{attribute 'reflection'}
PROGRAM SystemBase // system base program, from here all modules are controlled and the system functions are called.
VAR_INPUT // System configuration settings
	bIcfAirCheckPresent	: BOOL := TRUE; // System is not equiped with air pressure sensor 
END_VAR
VAR	// Fault indications
	bMissingCond		: BOOL := FALSE ; // Module missing condition active
	bFatalFault			: BOOL := FALSE ; // Module fatal fault is active
	bCycleFault			: BOOL := FALSE ; // Module cycle fault is active

	// Check values
	bReferenceOk		: BOOL := FALSE ; // All module references  have been checked

	// State indication
	bSafeStopping		: BOOL := FALSE ; // Module is stopping by safety
	bIsSafe				: BOOL := FALSE ; // Module is safe and locked until safety is ok
	bNoreference		: BOOL := FALSE ; // Module Startup Undefined initialization required

	bInitializing		: BOOL := FALSE ; // Module startup initializing
	bInitialized		: BOOL := FALSE ; // Module startup initialized waiting for startup command
	
	bParametersLoaded 	: BOOL := FALSE ; // Parameters have been loaded from the file(s) 

	bIdle 				: BOOL := FALSE ; // Module startup Idle no commands active

	bEnabling 			: BOOL := FALSE ; // Module Startup enabeling 
	bEnabled 			: BOOL := FALSE ; // Module Startup Enabled
	
	bHoming				: BOOL := FALSE ; // Module startup homing back to base position and recalibrate
	bHomed 				: BOOL := FALSE ; // Module startup homed waiting for further further commands

	bHolding 			: BOOL := FALSE ; // Module Module Hold motion command executing
	bHeld	 			: BOOL := FALSE ; // Module Hold Motion is held until command is released	
	
	bResetting 			: BOOL := FALSE ; // Module Reset resetting error status
	bResetDone 			: BOOL := FALSE ; // Module reset is done   

	bManual 			: BOOL := FALSE ; // Module Work status Module in Manual 
	
	bStartSemiAuto		: BOOL := FALSE ; // Start semi automatic mode 
	bSemiAuto			: BOOL := FALSE ; // Module work status module in semi automatic
	
	bStartAuto			: BOOL := FALSE ; // Start automatic mode
	bAutomatic 			: BOOL := FALSE ; // Module Work status Module in Automatic mode
	bStopAuto			: BOOL := FALSE ; // Start automatic mode
	bStoppingAuto		: BOOL := FALSE ; // Start automatic mode
	
	bCmdPause			: BOOL := FALSE ; // Pause all modules 
	bPaused 			: BOOL := FALSE ; // all modules are paused
	
	bPoweringOff		: BOOL := FALSE ; // Module is powering off
	bPoweredOff			: BOOL := FALSE ; // Module has powered off 	

	bModuleLocked		: BOOL := FALSE ; // a module is locked for commands
	
	bAckWarningsBusy	: BOOL := FALSE	; // The acknowledge process is busy
END_VAR
VAR
	// System inputs 
	ibPowerSupplyOk	 	AT%I*	: BOOL  ; // System Power supply is ok 
	iSystemSafetyFault	AT%I*	: BOOL	; // System safety Fault
	fbAirpressureOk 			: Fb_DevDigitalInputFunctions  	; // system airpressure is ok
	fbCmdResetSafety		 	: FB_DevPushbuttonLight 		; // System reset
	
	fTrigPowerSupply			: F_TRIG ; // falling edge trigger for power supply
	toffMainAir					: TOF	:= (PT := T#500MS ); // Main air supply off delay
	// System safety valve
	fbValveMainAirSupply		: FB_DevValve ; // Main air supply valve 
	
	// System HMI commands
	fbStartSemiAuto				: FB_DevHMIButton ; // HMI start semi automatic button 
	fbStartAuto					: FB_DevHMIButton ; // HMI start automatic button
	fbResetSystem				: FB_DevHMIButton ; // HMI Reset system
	fbCmdPowerOff				: FB_DevHMIButton ; // HMI Power off system
	fbAckWarning				: FB_DevHMIButton ; // HMI Acknowledge warnings

	// system Commands 
	fbCmdStartSystem		 	: FB_DevPushbuttonLight  		; // (re)start system input from button
	fbCmdStartAuto				: FB_DevPushbuttonLight			; // Start system automatic cycle
	fbCmdStopAuto				: FB_DevPushbuttonLight			; // Start system automatic cycle
	
	//System state
	bSafetyOK					: BOOL := FALSE ;
	bAirOk						: BOOL := FALSE ; // Air pressure is ok 
	bSystemOK					: BOOL := FALSE ; // all safety and vitals are OK
	eStateSystem				: E_StateSystem := E_StateSystem.NoReference ; // State of system
	
	// Set system variables
	fbSetSystemVariables		: Fb_SystemVariables ;
	
	// System Fault handling
//	fbSystemFaultHandler		: Fb_SystemFaultHandler ;
//	fbOperatorMessage			: FB_OperatorMessageDisplay ; //Operator message or system state message hadler 

	// Local Fault Handling
	stFault					: UDT_Fault			; // Message data

 	// Module states
	nNumberOfModules			: UDINT := 0 ; // Number of modules added to the system 
	arpModules					: ARRAY [1..gvl_main.cnMaxNUMBEROFMODULES] OF Udt_ModuleId ; 

	// power down system function
	ntShutDown					: NT_Shutdown ; // shutdown system function 

	// Manual controller
	bDevicesAddedtoManual 		: BOOL := FALSE ; // Add system device (buttons) to manual controller
	

	// Function path 
	{attribute 'instance-path'} 
    {attribute 'noinit'}
	sPath			: STRING	; // Path name of function (used for manual reference
END_VAR
VAR // safety 
	// inputs 
	ibEstopOk 			AT%I*	: BOOL  ; // system emergency stop ok
	ibSystemSafetyOK	AT%I*	: BOOL  ; // System is safe 
	iSafetyFBErr		AT%I*	: BOOL	; // The "FB Error" group signal
	iSafetyComErr		AT%I*	: BOOL	; // The "Com Error" group signal
	iSafetyOtherErr		AT%I*	: BOOL	; // The "Other Err" group signal
	iSafetyOutErr		AT%I*	: BOOL	; // The "Out Err" group signal
	iSTOFault			AT%I* 	: BOOL	; // Motor safe torque off fault active
	
	// Outputs 
	qbSafetyErrAckn		AT%Q*	: BOOL ; // Safety error acknowledge
	qbRunSafety			AT%Q*	: BOOL ; // Run safety program
	qbResetSafety		AT%Q*	: BOOL ; // reset safety program
	qbSTOErrAckn		AT%Q*	: BOOL ; // Safet torque off error acnowledge

	// safety Reset Timer	
	TofSafetyErrAck				: TOF := (PT := T#500MS); // Safety reset timer
	TOfSTOErrAck				: TOF := (PT := T#500MS); // Safe torque off rest timer
END_VAR
VAR // Miscellaneous
	bFirstCycle : BOOL := TRUE; // Is this the first time the PRG is called?
	bPersistentDataFail	: BOOL := TRUE ;
END_VAR
VAR PERSISTENT // Persistent data check
	bPersistentFlag	: BOOL := FALSE ; // Persistent dat in tack flag
END_VAR

// Exec safety control
ExecSafetyControl();

// Call faulthandler
//fbSystemFaultHandler( 	nNumberOfModules	:= nNumberOfModules,
//						arpModules			:= arpModules,
//						bsystemInitialized	:= bInitialized,
//						bSystemFF			=> bFatalFault,
//						bSystemCF			=> bCycleFault,
//						bSystemMC			=> bMissingCond);

// Check if this is the first cycle the PRG is called
// if not, return. This is to make sure all modules are connected. 
IF bFirstCycle THEN
	bFirstCycle := FALSE;
	RETURN;
END_IF

// check system functions
IF bInitialized THEN 
	CheckSystemOK();
	CheckSystemCommands();
END_IF 

// Run system
ExecSystemRun();

// call device functions 
CallSystemFunctions();

// Call operator warning acknowledgement
ExecAckWarnings();

// Call modules 
CallModules();

METHOD PRIVATE CallModules : BOOL
VAR
	i : UDINT ;
END_VAR
VAR
	AllAutomatic : BOOL ;
	
	Stopping : BOOL;
	bAllStopped : BOOL;
END_VAR
// set base conditions
bReferenceOk	:= TRUE ;
bIsSafe			:= TRUE ;
bIdle			:= TRUE ;	
bHeld			:= TRUE ;
bResetDone 		S= bResetting	;
bManual			:= TRUE	;
bSemiAuto		:= TRUE ;
bAutomatic		:= FALSE; // Reverse feedback 
AllAutomatic 	:= TRUE ;
bStoppingAuto	:= TRUE ;
bEnabled		S= bEnabling ;
bPoweredOff		:= TRUE;
bHomed 			:= TRUE;
bPaused 		:= TRUE;
bAllStopped     := TRUE;

// copy inputs to modules 
FOR i := 1 TO nNumberOfModules DO 
	// set system commands
	arpModules[i].pFunction^.bEnable			:= bEnabled			;
	arpModules[i].pFunction^.bCmdReset			:= bResetting		;
	arpModules[i].pFunction^.bSafetyOK			:= NOT bSafeStopping;
	arpModules[i].pFunction^.bCmdPause			:= bCmdPause		; 
	// Read state indications 
	bReferenceOk 	:= arpModules[i].pFunction^.bReferenceOk 	AND bReferenceOk; 
	bIsSafe 		:= arpModules[i].pFunction^.bIsSafe 		AND bIsSafe		;
	bEnabled 		:= arpModules[i].pFunction^.bEnable 		AND bEnabled	;
	bHeld			:= arpModules[i].pFunction^.bHeld 			AND bHeld		;
	bResetDone		:= arpModules[i].pFunction^.bResetDone 		AND bResetDone	;
	bManual			:= arpModules[i].pFunction^.bManual 		AND bManual		;
	bSemiAuto		:= arpModules[i].pFunction^.bSemiAuto 		AND bSemiAuto	;
	bPoweredOff 	:= arpModules[i].pFunction^.bPoweredOff 	AND bPoweredOff	;
	bHomed			:= arpModules[i].pFunction^.bHomed			AND bHomed 		;
	bPaused			:= arpModules[i].pFunction^.bPaused			AND bPaused		;
	bModuleLocked	S= arpModules[i].pFunction^.bLocked							; // Module is locked for commnds
	bCmdPause 		R= arpModules[i].pFunction^.bReqContinue					; // Request continue from module
	bCmdPause		S= arpModules[i].pFunction^.bReqPause						; // Request for pause from module
	bAutomatic		S= arpModules[i].pFunction^.bAutomatic 						; // Stay in automatic even when one module is in automatic
	AllAutomatic	:= arpModules[i].pFunction^.bAutomatic 		AND AllAutomatic; // reset start automatic when al modules are in automatic operation
	bStoppingAuto	:= arpModules[i].pFunction^.bStopping 		AND bStoppingAuto; // reset start automatic when al modules are in automatic operation

	Stopping		:= arpModules[i].pFunction^.bStopping;
	
	bAllStopped     := NOT Stopping AND NOT bAutomatic AND bAllStopped;

	
END_FOR

// Reset start inputs
	bEnabling		R= bEnabled 	;
	bHolding		R= bHeld 		;
	bResetting		R= bResetDone 	;
	bStartSemiAuto	R= bSemiAuto	;
	bPoweringOff	R= bPoweredOff 	;
	bHoming			R= bHomed 		;
	bStartAuto		R= AllAutomatic	; 
	bStopAuto		R= bAllStopped	;
	bCmdPause		R= NOT bAutomatic	;
END_METHOD

METHOD PRIVATE CallSystemFunctions : BOOL
VAR_INPUT
END_VAR
// call parameter handler
GVL_Parameters.fbParameterHandler();
IBF_Devices.GVL_DevManual.fbManualControler();

// Execute button functions 
fbStartAuto		( 	tDelay			:= T#100MS,
					refFbManualCtrl	:= IBF_Devices.GVL_DevManual.fbManualControler);
fbStartSemiAuto ( 	tDelay			:= T#100MS,
					refFbManualCtrl	:= IBF_Devices.GVL_DevManual.fbManualControler); 
fbResetSystem 	( 	tDelay			:= T#5000MS,
					refFbManualCtrl	:= IBF_Devices.GVL_DevManual.fbManualControler); 
//fbAckWarning	(	Istatus			:= GVL_Message.bAckWarnings,
//					tDelay			:= T#100MS,
//					refFbManualCtrl := IBF_Devices.GVL_DevManual.fbManualControler,
//					refFbFault 		:= fbFaultHandler );

fbCmdStartSystem(	refFbManualCtrl	:= IBF_Devices.GVL_DevManual.fbManualControler);
fbCmdStartAuto	(	refFbManualCtrl	:= IBF_Devices.GVL_DevManual.fbManualControler);
fbCmdStopAuto	(	refFbManualCtrl	:= IBF_Devices.GVL_DevManual.fbManualControler);

// execute input functions
fbValveMainAirSupply(	bEnable			:= TRUE,
						bSafetyOk		:= ibEstopOk,
						refFbManualCtrl	:= IBF_Devices.GVL_DevManual.fbManualControler);

// Add device functions to manual controller 
IF NOT bDevicesAddedtoManual THEN
	IF bIcfAirCheckPresent THEN
		IBF_Devices.GVL_DevManual.fbManualControler.CmdAddDevice( refToDevice := fbAirpressureOk 	);
	END_IF
	IBF_Devices.GVL_DevManual.fbManualControler.CmdAddDevice( refToDevice := fbCmdStartSystem	);
	IBF_Devices.GVL_DevManual.fbManualControler.CmdAddDevice( refToDevice := fbCmdStartAuto		);
	IBF_Devices.GVL_DevManual.fbManualControler.CmdAddDevice( refToDevice := fbCmdStopAuto		);
	IBF_Devices.GVL_DevManual.fbManualControler.CmdAddDevice( refToDevice := fbCmdResetSafety	);
	bDevicesAddedtoManual S= TRUE ;
END_IF
END_METHOD

METHOD INTERNAL CheckSystemCommands : BOOL
VAR_INPUT
END_VAR
// ===== full reset ======
	IF fbCmdResetSafety.bFcoDelay THEN 
		eStateSystem 	:= E_StateSystem.NoReference ;
	END_IF

// ====== power off ======
	IF fbCmdPowerOff.bFcoDelay THEN 
		eStateSystem := E_StateSystem.PowerOff ;
	END_IF
END_METHOD

METHOD PRIVATE CheckSystemOK : BOOL
// shutdown emediately if power is down 
fTrigPowerSupply(CLK := ibPowerSupplyOk);
ntShutDown(START := GVL_Main.cbUPSPRESENT AND (bPoweredOff OR fTrigPowerSupply.Q)); 

// ===== Check Air pressure =====
IF bIcfAirCheckPresent THEN
	fbAirpressureOk(refFbManualCtrl	:= IBF_Devices.GVL_DevManual.fbManualControler);
	bAirOk := fbAirpressureOk.bFcoDelay ;
ELSE
	bAirOk := TRUE ;
END_IF


// ===== Check if system is ok =====
	bSystemOK := TRUE ;
	bSystemOK := bAirOk 	AND bSystemOK ;
	bSystemOK := bSafetyOK	AND bSystemOK ;	
				
	IF NOT bSystemOK 
	AND eStateSystem > E_StateSystem.Safe 
	AND eStateSystem <> E_StateSystem.Resetting 
	THEN
		eStateSystem := E_StateSystem.Safe; 
	ELSIF (bFatalFault OR bCycleFault) 
	AND eStateSystem <> E_StateSystem.Resetting 
	THEN 
		eStateSystem := E_StateSystem.Fault ;
	END_IF

// ===== System messages ======
	IF NOT bAirOk THEN
		stFault.Active 		:= TRUE ;
		stFault.Description	:= 'Main air Pressure low ';
		stFault.FaultType		:= E_FaultTypes.FF;
		IBF_HMI.GVL_HMI.fbHMIControl.bShowEmergencyOverlay := TRUE;
		IBF_HMI.GVL_HMI.fbHMIControl.sEmergencyText := 'AIR PRESSURE LOW';
	END_IF
	
// Main air control 
toffMainAir(IN := bSystemOK);
IF toffMainAir.Q THEN
	fbValveMainAirSupply.CmdOpen();
END_IF
END_METHOD

METHOD PUBLIC CmdAddModule : BOOL
VAR_INPUT
	refToModule : REFERENCE TO Fb_ModuleBase ; // reference to module function
END_VAR
VAR
	bModuleAdded	: BOOL := FALSE;
	i 				: UDINT ; 
END_VAR
// Check if device is not already in the array 
FOR i:= 1 TO GVL_Main.cnMaxNUMBEROFMODULES DO
	IF arpModules[i].pFunction = 0 THEN 
		nNumberOfModules:= i;
		EXIT;	
	ELSIF arpModules[i].sName = refToModule.stIdentity.sName THEN 
		bModuleAdded := TRUE ;
	END_IF 
END_FOR

// If device is not found add device to the list
IF NOT bModuleAdded AND nNumberOfModules >= 1 AND nNumberOfModules <= GVL_Main.cnMaxNUMBEROFMODULES THEN
	arpModules[nNumberOfModules].nNumber 	:= refToModule.nModuleID;
	arpModules[nNumberOfModules].sName		:= refToModule.stIdentity.sName	;
	arpModules[nNumberOfModules].pFunction 	:= ADR(refToModule)		;	
	bModuleAdded := TRUE ;
END_IF

CmdAddModule := bModuleAdded ;
END_METHOD

METHOD CmdReset : BOOL
VAR_INPUT
END_VAR
eStateSystem := E_StateSystem.Resetting;

CmdReset := TRUE;
END_METHOD

METHOD ExecAckWarnings : BOOL
VAR
	i : UDINT ;
END_VAR
//If required, run the acknowledge process 
IF (fbAckWarning.bFeStatus OR NOT bAckWarningsBusy) THEN
	bAckWarningsBusy := TRUE;
	
	FOR i := 1 TO nNumberOfModules DO 
		bAckWarningsBusy := arpModules[i].pFunction^.CmdAckOW() AND bAckWarningsBusy;
	END_FOR
END_IF
END_METHOD

METHOD PRIVATE ExecAutomatic : BOOL
VAR_INPUT
END_VAR
VAR
	i : UDINT ;
END_VAR
IF bStopAuto THEN 
	FOR i := 1 TO nNumberOfModules DO 
		arpModules[i].pFunction^.CmdStopAutomatic() ;
	END_FOR
ELSIF bStartAuto THEN 
	// Run automatic function in 
	FOR i := 1 TO nNumberOfModules DO 
		arpModules[i].pFunction^.CmdAutomatic() ;
	END_FOR
END_IF
	
ExecAutomatic := NOT bStartAuto;
END_METHOD

METHOD PRIVATE ExecHoming : BOOL
VAR_INPUT
END_VAR
VAR
	i : UDINT ;
END_VAR
// Home all modules
FOR i := 1 TO nNumberOfModules DO 
	IF NOT arpModules[i].pFunction^.bHomed THEN 
		arpModules[i].pFunction^.CmdHome();
	END_IF
END_FOR
 
bHoming := NOT bHomed;
ExecHoming := bHomed;
END_METHOD

METHOD PUBLIC ExecManual : BOOL
VAR
	i : UDINT ;
END_VAR
bEnabled := FALSE ;
// Run automatic function in 
FOR i := 1 TO nNumberOfModules DO 
	arpModules[i].pFunction^.CmdManual() ;
END_FOR

ExecManual := bManual;
END_METHOD

METHOD PRIVATE ExecPowerOff : BOOL
VAR_INPUT
END_VAR
VAR 
	i : UDINT ;
END_VAR
// Power off all modules
FOR i := 1 TO nNumberOfModules DO 
	arpModules[i].pFunction^.CmdPowerOff () ;
END_FOR
 
ExecPowerOff := bPoweredOff ;
END_METHOD

METHOD PRIVATE ExecSafeHold : BOOL
VAR_INPUT
END_VAR
VAR
	i : UDINT ;
END_VAR
// Hold all modules
bStartAuto		:= FALSE;

FOR i := 1 TO nNumberOfModules DO 
	arpModules[i].pFunction^.CmdHold();
END_FOR

ExecSafeHold := bHeld ;
END_METHOD

METHOD PRIVATE ExecSafeReset : BOOL
VAR_INPUT
END_VAR
END_METHOD

METHOD PRIVATE ExecSafeStop : BOOL
VAR_INPUT
END_VAR
VAR
	i : UDINT ;
END_VAR
bEnabling		:= FALSE;
bInitializing	:= FALSE;
bHoming			:= FALSE;
bStartAuto		:= FALSE;
bStartSemiAuto	:= FALSE;

// Module safe stop
IF bInitialized AND bReferenceOk THEN 
	FOR i := 1 TO nNumberOfModules DO 
		arpModules[i].pFunction^.CmdEstop();
	END_FOR
END_IF

IF bIsSafe THEN 
	fbValveMainAirSupply.CmdSafeStop();
END_IF
 
ExecSafeStop := bIsSafe ;
END_METHOD

METHOD PRIVATE ExecSafetyControl : BOOL
VAR_INPUT
END_VAR
IF ibEstopOk 
AND ibSystemSafetyOK
AND NOT iSTOFault
THEN
	bSafetyOK				S= TRUE ;
	IBF_HMI.GVL_HMI.fbHMIControl.bShowEmergencyOverlay	:= FALSE ;
ELSE 
	bSafetyOK				:= FALSE ;
	IBF_HMI.GVL_HMI.fbHMIControl.bShowEmergencyOverlay	:= TRUE ;
	IF eStateSystem > E_StateSystem.Safe 
	AND eStateSystem <> E_StateSystem.Resetting  THEN 
		eStateSystem			:= E_StateSystem.Safe ;
	END_IF
END_IF

// Set safety state and button light state
fbCmdResetSafety.bEnable S= TRUE ;
IF NOT ibEstopOk THEN 
	IBF_HMI.GVL_HMI.fbHMIControl.bShowEmergencyOverlay	:= TRUE ;
	fbCmdResetSafety.CmdOn() ;
ELSIF NOT ibSystemSafetyOK OR iSTOFault THEN 
	fbCmdResetSafety.CmdBlinkSlow() ;
ELSIF NOT bAirOk OR NOT bSystemOK THEN
	fbCmdResetSafety.CmdBlinkFast() ;
END_IF



// Safety reset button function
fbCmdResetSafety(	tDelay			:= T#30S ,
					refFbManualCtrl	:= IBF_Devices.GVL_DevManual.fbManualControler); 

// Link safety reset
qbResetSafety := fbCmdResetSafety.bFeStatus AND NOT bSafetyOK ;

// Set safety system in run mode
IF NOT iSafetyFBErr 
AND NOT iSafetyComErr
AND NOT iSafetyOtherErr
AND NOT iSafetyOutErr
AND NOT iSystemSafetyFault 
AND bInitialized THEN 
	qbRunSafety := TRUE ;
ELSE 
	qbRunSafety := FALSE;
END_IF

// reset safety faults
TofSafetyErrAck	(IN := qbSafetyErrAckn	);
TOfSTOErrAck	(IN := qbSTOErrAckn 	);
qbSTOErrAckn	:= FALSE ;
qbSafetyErrAckn := FALSE ;

IF iSafetyFBErr THEN 
	IBF_HMI.GVL_HMI.fbHMIControl.sEmergencyText 	:= 'Safety Program Function block error';
	IF NOT qbRunSafety AND NOT TofSafetyErrAck.Q THEN 
		qbSafetyErrAckn := TRUE; 
	END_IF
	stFault.Active := TRUE ;
	stFault.Description	:= 'Safety program is in fault state.';
	stFault.FaultType		:= E_FaultTypes.FF;

	IBF_HMI.GVL_HMI.fbHMIControl.sEmergencyText 	:= 'Safety program is in fault state.';
ELSIF iSafetyComErr THEN
	IBF_HMI.GVL_HMI.fbHMIControl.sEmergencyText 	:= 'Safety program com error';
	IF NOT qbRunSafety AND NOT TofSafetyErrAck.Q THEN 
		qbSafetyErrAckn := TRUE ;
	END_IF
	stFault.Active 		:= TRUE ;
	stFault.Description	:= 'Emergency stop fault, check emergency button wiring ';
	stFault.FaultType		:= E_FaultTypes.FF;
	IBF_HMI.GVL_HMI.fbHMIControl.sEmergencyText 	:= 'Emergency stop fault, check emergency button wiring ';
ELSIF iSafetyOutErr THEN
	IBF_HMI.GVL_HMI.fbHMIControl.sEmergencyText 	:= 'Safety program out error';
	IF NOT qbRunSafety AND NOT TofSafetyErrAck.Q THEN 
		qbSafetyErrAckn := TRUE ;
	END_IF
	stFault.Active 		:= TRUE ;
	stFault.Description	:= 'Emergency stop fault, check wiring ';
	stFault.FaultType		:= E_FaultTypes.FF;
	IBF_HMI.GVL_HMI.fbHMIControl.sEmergencyText 	:= 'Emergency stop fault, check wiring ';
ELSIF iSafetyOtherErr THEN
	IBF_HMI.GVL_HMI.fbHMIControl.sEmergencyText 	:= 'Safety program other error';
	IF NOT qbRunSafety AND NOT TofSafetyErrAck.Q THEN 
		qbSafetyErrAckn := TRUE ;
	END_IF
	stFault.Active 		:= TRUE ;
	stFault.Description	:= 'Safety program is in fault state. ';
	stFault.FaultType		:= E_FaultTypes.FF;
	IBF_HMI.GVL_HMI.fbHMIControl.sEmergencyText 	:= 'Safety program is in fault state. ';
ELSIF iSystemSafetyFault THEN
// System safety function faults 
	IBF_HMI.GVL_HMI.fbHMIControl.sEmergencyText 	:= 'Collision detection fault, check sensor wiring';
	IF NOT qbRunSafety AND NOT TofSafetyErrAck.Q THEN 
		qbSafetyErrAckn := TRUE ;
	END_IF
	stFault.Active 		:= TRUE ;
	stFault.Description	:= 'Collision safety fault, check collision detection wiring ';
	stFault.FaultType		:= E_FaultTypes.FF;
	IBF_HMI.GVL_HMI.fbHMIControl.sEmergencyText 	:= 'System safety fault, check wiring ';
ELSIF iSTOFault THEN
	IBF_HMI.GVL_HMI.fbHMIControl.sEmergencyText 	:= 'Motor safety fault';
	qbSTOErrAckn 			:= Sys_Variables.HeartBeat ;
	stFault.Active 		:= TRUE ;
	stFault.Description	:= 'Collision safety fault, check collision detection wiring ';
	stFault.FaultType		:= E_FaultTypes.FF;
	IBF_HMI.GVL_HMI.fbHMIControl.sEmergencyText 	:= 'Motor safe torque off fault';
ELSIF NOT ibEstopOk THEN
	IBF_HMI.GVL_HMI.fbHMIControl.sEmergencyText 	:= 'Emergency stop pressed';
ELSIF NOT ibSystemSafetyOK THEN 
	IBF_HMI.GVL_HMI.fbHMIControl.sEmergencyText 	:= 'Safety bumper pressed';
END_IF
END_METHOD

METHOD PUBLIC ExecSemiAuto : BOOL
VAR
	i : UDINT ;
END_VAR
// Run automatic function in 
FOR i := 1 TO nNumberOfModules DO 
	arpModules[i].pFunction^.CmdSemiAuto() ;
END_FOR

ExecSemiAuto := bSemiAuto;
END_METHOD

METHOD INTERNAL ExecSystemRun : BOOL
VAR_INPUT
END_VAR
// set system variables 
fbSetSystemVariables();

// State machine 
CASE eStateSystem OF 
	E_StateSystem.NoReference:
		IBF_HMI.GVL_HMI.fbHMIControl.eHomeScreen := E_BaseVisu.Idle;
		bHomed			:= FALSE ;
		bEnabled		:= FALSE ;
		IF bReferenceOk THEN
			eStateSystem 	:= E_StateSystem.Initialize ;
		END_IF
	E_StateSystem.Initialize:
		IF Init() THEN
			eStateSystem := E_StateSystem.LoadParameters;
		END_IF
	E_StateSystem.LoadParameters:
		bParametersLoaded := GVL_Parameters.fbParameterHandler.Init(); 
		IF bParametersLoaded OR GVL_Parameters.fbParameterHandler.bFault THEN
			eStateSystem := E_StateSystem.Safe ;
		END_IF
	E_StateSystem.Safe:
		bSafeStopping := NOT bIsSafe;
		IF bIsSafe 
		AND bSystemOK THEN 
			IF bFatalFault OR bCycleFault THEN
				eStateSystem := E_StateSystem.Fault ;
			ELSE
				eStateSystem := E_StateSystem.Enable;
			END_IF
		ELSIF fbResetSystem.bFeStatus THEN
			eStateSystem	:= E_StateSystem.Resetting;
		ELSE 
			ExecSafeStop();
		END_IF
	E_StateSystem.Enable:
		bEnabling 	:= bSystemOK;
		IF GVL_HMI.fbHMIControl.bInScreenManual THEN
			eStateSystem := E_StateSystem.Manual ;
		ELSIF bEnabled THEN 
			fbCmdStartSystem.CmdBlinkFast();
			IF fbCmdResetSafety.bFeStatus THEN
				eStateSystem := E_StateSystem.Resetting ;
			ELSIF fbCmdStartSystem.bFeStatus THEN
				eStateSystem := E_StateSystem.Home ;
			END_IF
		END_IF
	E_StateSystem.Home:	
		IF fbCmdResetSafety.bFeStatus THEN
			eStateSystem := E_StateSystem.Safe;			
		ELSIF ExecHoming() THEN
			eStateSystem := E_StateSystem.Idle;
		END_IF
	E_StateSystem.Resetting:
		IF NOT bResetDone THEN 
			bResetting S= TRUE ;
		ELSIF NOT bSafetyOK THEN 
			eStateSystem := E_StateSystem.Safe ;
		ELSIF bFatalFault OR bCycleFault THEN
			eStateSystem := E_StateSystem.Fault ;
		ELSIF bHomed THEN
			eStateSystem := E_StateSystem.Idle ;
		ELSE 
			eStateSystem := E_StateSystem.Enable ;
		END_IF
	E_StateSystem.Idle:
		fbCmdStartSystem.CmdBlinkSlow();
		IF fbCmdResetSafety.bFeStatus OR fbResetSystem.bFeStatus THEN
			eStateSystem := E_StateSystem.Resetting;			
		ELSIF GVL_HMI.fbHMIControl.bInScreenManual THEN 
			eStateSystem := E_StateSystem.Manual ;
		ELSIF bSystemOK AND fbCmdStartSystem.bFeStatus THEN 
			eStateSystem := E_StateSystem.SemiAuto ;
		END_IF
	E_StateSystem.Manual:
		IF fbCmdResetSafety.bFeStatus THEN
			eStateSystem := E_StateSystem.Safe;			
		ELSIF IBF_Devices.GVL_DevManual.bManualModeActive THEN
			ExecManual();
		END_IF
		
		IF NOT GVL_HMI.fbHMIControl.bInScreenManual THEN
			EStateSystem := E_StateSystem.Enable;
		END_IF 
	E_StateSystem.SemiAuto:
		ExecSemiAuto();
		IBF_HMI.GVL_HMI.fbHMIControl.eHomeScreen := E_BaseVisu.SemiAutomatic;
		IF fbCmdResetSafety.bFeStatus THEN
			eStateSystem := E_StateSystem.Idle;			
		ELSIF (fbCmdStartAuto.bFeStatus 
		OR fbStartAuto.bFcoDelay 
		OR bAutomatic)
		AND NOT bModuleLocked THEN 
			bStartAuto 		:= TRUE ;
			bStopAuto 		:= FALSE;
			eStateSystem 	:= E_StateSystem.Automatic ;
		END_IF					
	E_StateSystem.Automatic:
		ExecAutomatic();
		IBF_HMI.GVL_HMI.fbHMIControl.eHomeScreen := E_BaseVisu.Automatic;
		IF fbCmdResetSafety.bFeStatus THEN
			eStateSystem := E_StateSystem.Safe;
		ELSIF bAutomatic THEN
			IF fbCmdStartSystem.bFeStatus THEN
				eStateSystem := E_StateSystem.Idle ;
			ELSIF fbCmdStopAuto.bFeStatus THEN
				bStopAuto := TRUE;
			ELSIF fbCmdStartAuto.bFeStatus OR bMissingCond THEN  
				bCmdPause 	:= NOT bPaused ;
			END_IF
		ELSIF NOT bStartAuto AND NOT bStopAuto THEN 
			eStateSystem := E_StateSystem.SemiAuto ;
		END_IF
		
		// Start button light control
		IF bAutomatic THEN 
			fbCmdStartAuto.CmdOn();
		ELSE
			fbCmdStartAuto.CmdBlinkFast(); 				
		END_IF
	E_StateSystem.Fault:
		IF fbResetSystem.bFeStatus OR fbCmdResetSafety.bFeStatus THEN
			bResetDone		:= FALSE ;
			eStateSystem 	:= E_StateSystem.Resetting ;
		ELSIF bFatalFault THEN 
			ExecSafeStop();
		ELSIF bCycleFault THEN 
			ExecSafeHold();	
		END_IF 
	E_StateSystem.PowerOff:
		ExecPowerOff();
	ELSE 
		;		
END_CASE

bModuleLocked := FALSE ;

IBF_HMI.GVL_HMI.fbHMIControl.sStatusText := TO_STRING(eStateSystem);
END_METHOD

METHOD PRIVATE Init : BOOL
VAR_INPUT
END_VAR
VAR
	i : UDINT ;
END_VAR
// initialize system functions
IF bIcfAirCheckPresent THEN
	fbAirpressureOk.Init	( 	nId 		:= 1,
								nParentId	:= 0 );
END_IF 

fbCmdResetSafety.Init	(	nId 		:= 2,
							nParentId	:= 0 );

fbValveMainAirSupply.Init(	nId			:= 3,
							nParentId	:= 0,
							eResetState	:= E_ValveResetState.Res_Closed,
							eSafeState	:= E_ValveResetState.Res_Closed);

fbCmdStartSystem.Init	( 	nId 		:= 4,
							nParentId	:= 0 );

fbCmdStartAuto.Init		( 	nId 		:= 5,
							nParentId	:= 0 );

fbCmdStopAuto.Init		( 	nId 		:= 6,
							nParentId	:= 0 );
							
// Initialize all modules
bInitialized	:= TRUE ;
FOR i := 1 TO nNumberOfModules DO 
	IF NOT arpModules[i].pFunction^.bInitialized THEN 
		arpModules[i].pFunction^.CmdInit();
	END_IF
	bInitialized 	:= bInitialized AND arpModules[i].pFunction^.bInitialized;
 END_FOR
 
bInitializing 	:= NOT bInitialized ;
Init := bInitialized ;
END_METHOD

END_PROGRAM

(* stored: Version 1.1.0.1, ProductVersion 3.1.4024.11
   POU SystemBase: Id {147e2f75-a8ca-43e4-acf3-ce2169ee9c02}, SpecialFunc None
   Folder ModuleFunctions: Id {fb1414af-f6e5-4202-8989-256aa0d1eacc}
   Folder SystemFunction: Id {05994c64-d0aa-4e7d-8ae3-f139ae256daf}
   Method CallModules: Id {7e8c963f-d98c-43d0-a3ed-11f16c2d5b4d}
   Method CallSystemFunctions: Id {5be4e1d6-b194-4082-99a1-645b475d1410}
   Method CheckSystemCommands: Id {7c2b1772-f51e-4aa3-a97a-1e93dcc6a18d}
   Method CheckSystemOK: Id {b3d7881d-8420-47b1-9d4b-1c3829d8822d}
   Method CmdAddModule: Id {02c45d8a-a400-4bf9-96fe-fbe272a81730}
   Method CmdReset: Id {81a11f00-ce22-44b4-b332-2d4b7e3055ba}
   Method ExecAckWarnings: Id {86c6f5a0-b6fe-4448-9452-f04a9ea3021f}
   Method ExecAutomatic: Id {3c758811-81f1-42d1-83e5-646cc80a7b4f}
   Method ExecHoming: Id {345df0e0-469c-4aba-9303-ad14c7d3f6d3}
   Method ExecManual: Id {1eeb2405-fd6d-491e-8ef7-e639f5684ed3}
   Method ExecPowerOff: Id {b17ea916-e40f-4a32-a9b5-a5ade237754d}
   Method ExecSafeHold: Id {09e80f99-469c-4643-bf23-6284454a47bf}
   Method ExecSafeReset: Id {1f949173-b753-460e-b2f0-a3f94b7a8c12}
   Method ExecSafeStop: Id {231fd871-3511-471c-84e1-00de0d5b0d2d}
   Method ExecSafetyControl: Id {8ec10b67-53de-4590-9578-2159b6a13b3f}
   Method ExecSemiAuto: Id {d1439c2c-5160-4c2a-96fa-c7dd6421b071}
   Method ExecSystemRun: Id {504c7dee-e26b-448e-99d5-004a6dc8da1e}
   Method Init: Id {77ed26c7-8922-4741-8b27-ccc11849164f} *)
